// Implicitly generated code : DO NOT EDIT
FUNCTION CheckDivLInt : LINT
VAR_INPUT
	divisor:LINT;
END_VAR

// Implicitly generated code : Only an Implementation suggestion
IF divisor = 0 THEN
	CheckDivLInt:=1;
	GVL_Checks.dCheckDivLInt := GVL_Checks.dCheckDivLInt + 1;
	ADSLOGSTR(4,'Checks critical error - LINT variable divided by 0.','');
ELSE
	CheckDivLInt:=divisor;
END_IF

END_FUNCTION

(* stored: Version 1.1.0.1, ProductVersion 3.1.4024.12
   POU CheckDivLInt: Id {f59dd30b-73ea-4bd5-974c-0699274ce057}, SpecialFunc CheckDivInt64 *)
